// TIA Portal V19 export
FUNCTION "CallManualOperationLines_Unit2" : Void   // FC83, LAD
// stored: SetENOAutomatically false
   VAR_TEMP
      status : Array[0..30] of Word;   // Status of the configuration or line FC
      errorID : Array[0..30] of Word;   // Error ID of the configuration or line FC
   END_VAR
BEGIN

REGION Network 1: Unit 2 Equipment Module 1 Configuration
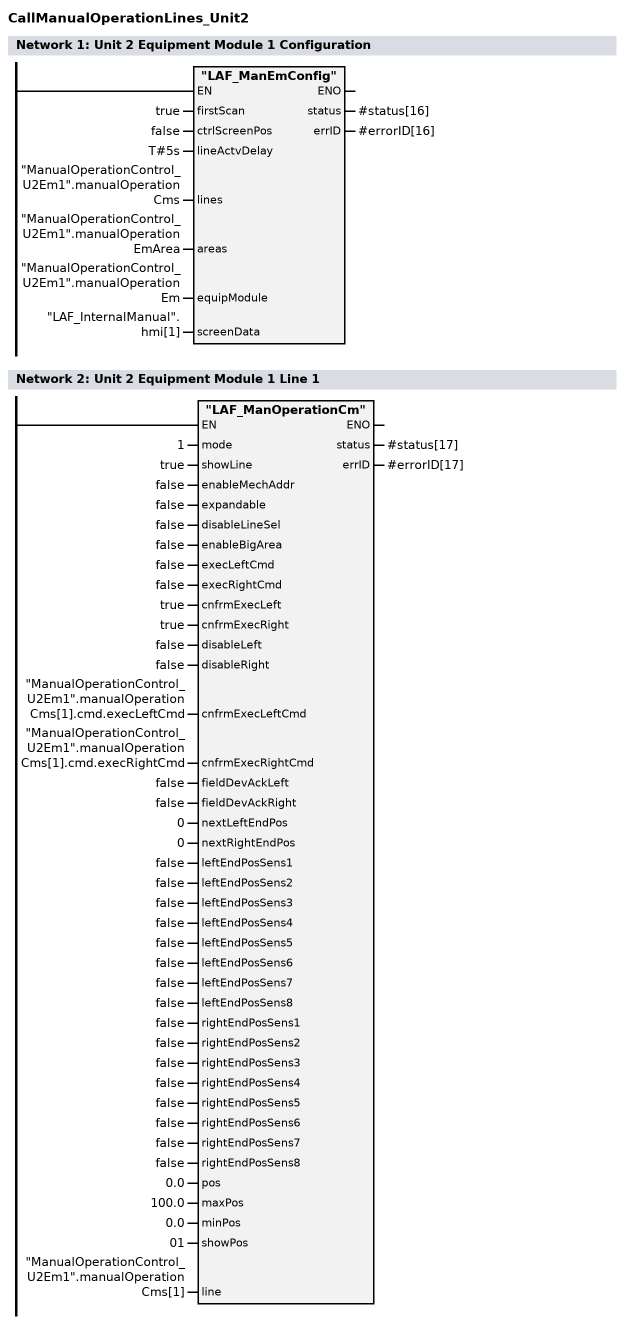
   RUNG wire#powerrail
      "LAF_ManEmConfig"(firstScan := true, ctrlScreenPos := false, lineActvDelay := T#5s, lines := "ManualOperationControl_U2Em1".manualOperationCms, areas := "ManualOperationControl_U2Em1".manualOperationEmArea, equipModule := "ManualOperationControl_U2Em1".manualOperationEm, screenData := "LAF_InternalManual".hmi[1], status => #status[16], errID => #errorID[16])
   END_RUNG
   // the same network as SCL:
   "LAF_ManEmConfig"(firstScan := true,
                     ctrlScreenPos := false,
                     lineActvDelay := T#5s,
                     lines := "ManualOperationControl_U2Em1".manualOperationCms,
                     areas := "ManualOperationControl_U2Em1".manualOperationEmArea,
                     equipModule := "ManualOperationControl_U2Em1".manualOperationEm,
                     screenData := "LAF_InternalManual".hmi[1],
                     status => #status[16],
                     errID => #errorID[16]);
END_REGION

REGION Network 2: Unit 2 Equipment Module 1 Line 1
   RUNG wire#powerrail
      "LAF_ManOperationCm"(mode := 1, showLine := true, enableMechAddr := false, expandable := false, disableLineSel := false, enableBigArea := false, execLeftCmd := false, execRightCmd := false, cnfrmExecLeft := true, cnfrmExecRight := true, disableLeft := false, disableRight := false, cnfrmExecLeftCmd := "ManualOperationControl_U2Em1".manualOperationCms[1].cmd.execLeftCmd, cnfrmExecRightCmd := "ManualOperationControl_U2Em1".manualOperationCms[1].cmd.execRightCmd, fieldDevAckLeft := false, fieldDevAckRight := false, nextLeftEndPos := 0, nextRightEndPos := 0, leftEndPosSens1 := false, leftEndPosSens2 := false, leftEndPosSens3 := false, leftEndPosSens4 := false, leftEndPosSens5 := false, leftEndPosSens6 := false, leftEndPosSens7 := false, leftEndPosSens8 := false, rightEndPosSens1 := false, rightEndPosSens2 := false, rightEndPosSens3 := false, rightEndPosSens4 := false, rightEndPosSens5 := false, rightEndPosSens6 := false, rightEndPosSens7 := false, rightEndPosSens8 := false, pos := 0.0, maxPos := 100.0, minPos := 0.0, showPos := 01, line := "ManualOperationControl_U2Em1".manualOperationCms[1], status => #status[17], errID => #errorID[17])
   END_RUNG
   // the same network as SCL:
   "LAF_ManOperationCm"(mode := 1,
                        showLine := true,
                        enableMechAddr := false,
                        expandable := false,
                        disableLineSel := false,
                        enableBigArea := false,
                        execLeftCmd := false,
                        execRightCmd := false,
                        cnfrmExecLeft := true,
                        cnfrmExecRight := true,
                        disableLeft := false,
                        disableRight := false,
                        cnfrmExecLeftCmd := "ManualOperationControl_U2Em1".manualOperationCms[1].cmd.execLeftCmd,
                        cnfrmExecRightCmd := "ManualOperationControl_U2Em1".manualOperationCms[1].cmd.execRightCmd,
                        fieldDevAckLeft := false,
                        fieldDevAckRight := false,
                        nextLeftEndPos := 0,
                        nextRightEndPos := 0,
                        leftEndPosSens1 := false,
                        leftEndPosSens2 := false,
                        leftEndPosSens3 := false,
                        leftEndPosSens4 := false,
                        leftEndPosSens5 := false,
                        leftEndPosSens6 := false,
                        leftEndPosSens7 := false,
                        leftEndPosSens8 := false,
                        rightEndPosSens1 := false,
                        rightEndPosSens2 := false,
                        rightEndPosSens3 := false,
                        rightEndPosSens4 := false,
                        rightEndPosSens5 := false,
                        rightEndPosSens6 := false,
                        rightEndPosSens7 := false,
                        rightEndPosSens8 := false,
                        pos := 0.0,
                        maxPos := 100.0,
                        minPos := 0.0,
                        showPos := 01,
                        line := "ManualOperationControl_U2Em1".manualOperationCms[1],
                        status => #status[17],
                        errID => #errorID[17]);
END_REGION
END_FUNCTION
